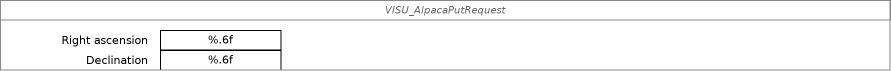
VISUALIZATION VISU_AlpacaPutSlewToCoordinates  // 891x71
VAR_IN_OUT
	stInstance : ST_AlpacaPutSlewToCoordinates;
END_VAR
    Frame (0,0 891x20)
        shows VISU_AlpacaPutRequest(stInstance := stInstance)
    Label (50,30 101x21), "Right ascension"
    Rectangle (160,30 121x20), "%.6f", text variable: stInstance.i_lrRightAscension
        OnMouseClick: write the text variable via Default
    Label (50,50 101x21), "Declination"
    Rectangle (160,50 121x20), "%.6f", text variable: stInstance.i_lrDeclination
        OnMouseClick: write the text variable via Default
END_VISUALIZATION

(* stored: Version 1.1.0.1, ProductVersion 3.1.4024.12
   Visu VISU_AlpacaPutSlewToCoordinates: Id {c24bc49c-2a3d-43e9-b3c6-883c718275f7} *)
